FUNCTION_BLOCK LuefterUeberwachung
VAR_INPUT
END_VAR
VAR_OUTPUT
END_VAR
VAR
END_VAR

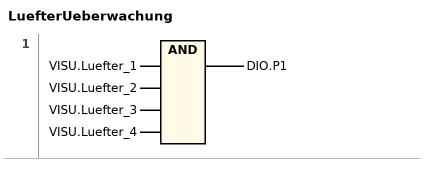
// NETWORK 1
DIO.P1 := VISU.Luefter_1 AND VISU.Luefter_2 AND VISU.Luefter_3 AND VISU.Luefter_4;

END_FUNCTION_BLOCK

(* stored: Version 1.1.0.1, ProductVersion 3.1.4022.6
   POU LuefterUeberwachung: Id {d266dc57-a678-43a7-8e11-96d978017ed9}, SpecialFunc None *)
